// TIA Portal V18 export
TYPE "LGasp_frenatura"
// stored: IsFailsafeCompliant false
   STRUCT
      nomeprogramma : WString[30];   // nome del programma della franatura da PC
      diametrocoilmax : LReal;   // diametro coil nuovo in mm da PC
      frenaturacoilmax : LReal;   // frenatura con coil massimo da PC
      diametrocoilmin : LReal;   // diametro mandrino vuoto mm da PC
      frenaturacoilmin : LReal;   // frenatura con coil minimo da PC
      velocita : LReal;   // riferimento di velocità durante frenatura
      diametrolaserattuale : LReal;   // diametro attuale rilevato dal laser da PLC
      coppiaattuale : LReal;   // coppia attuale motore da PLC
   END_STRUCT;
END_TYPE
